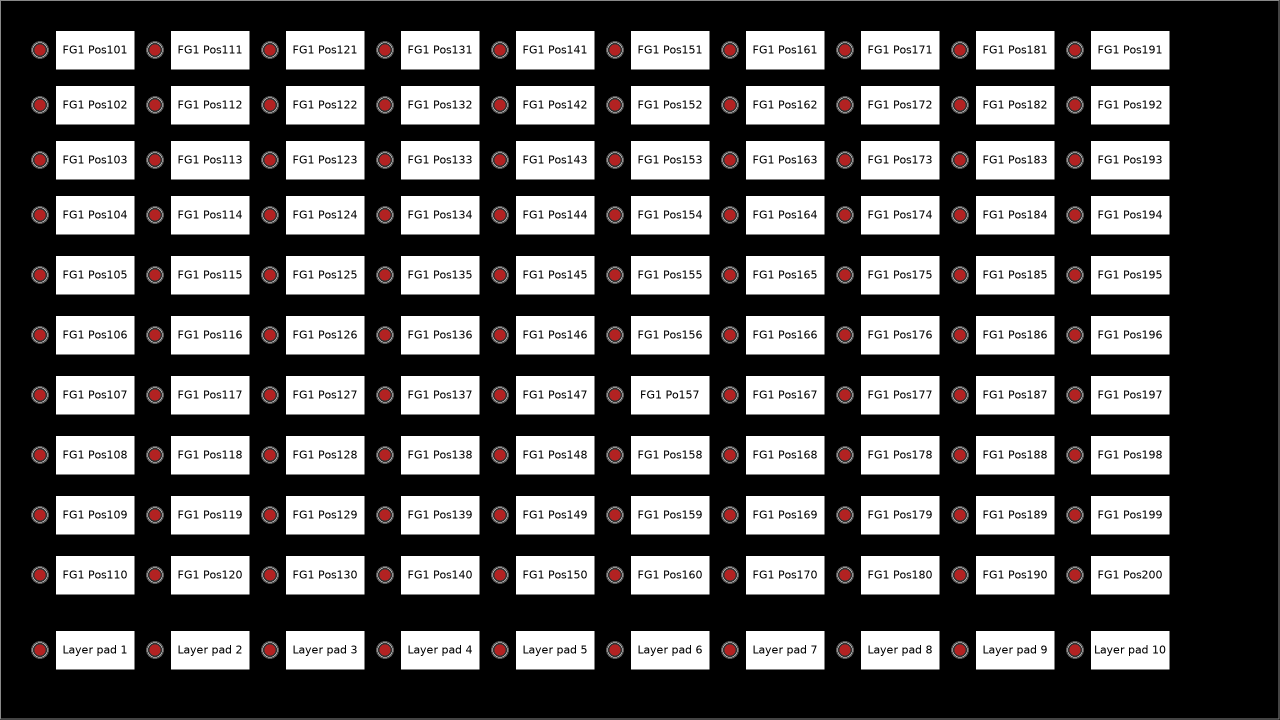
VISUALIZATION PAGE_KR1_Tab_1_200  // 1280x720
    RoundedRectangle (170,30 80x40), "FG1 Pos111"
        toggle KR1.bOutBit[18,0]
        OnMouseClick: execute {  }
    Lamp1 (145,40 20x20), variable: KR1.bInBit[18,0], style: Lamp-Lamp1-Red
    RoundedRectangle (55,30 80x40), "FG1 Pos101"
        toggle KR1.bOutBit[16,6]
        OnMouseClick: execute {  }
    Lamp1 (30,40 20x20), variable: KR1.bInBit[16,6], style: Lamp-Lamp1-Red
    RoundedRectangle (285,30 80x40), "FG1 Pos121"
        toggle KR1.bOutBit[19,2]
        OnMouseClick: execute {  }
    Lamp1 (260,40 20x20), variable: KR1.bInBit[19,2], style: Lamp-Lamp1-Red
    RoundedRectangle (400,30 80x40), "FG1 Pos131"
        toggle KR1.bOutBit[20,4]
        OnMouseClick: execute {  }
    Lamp1 (375,40 20x20), variable: KR1.bInBit[20,4], style: Lamp-Lamp1-Red
    RoundedRectangle (515,30 80x40), "FG1 Pos141"
        toggle KR1.bOutBit[21,6]
        OnMouseClick: execute {  }
    Lamp1 (490,40 20x20), variable: KR1.bInBit[21,6], style: Lamp-Lamp1-Red
    RoundedRectangle (745,30 80x40), "FG1 Pos161"
        toggle KR1.bOutBit[24,2]
        OnMouseClick: execute {  }
    Lamp1 (720,40 20x20), variable: KR1.bInBit[24,2], style: Lamp-Lamp1-Red
    RoundedRectangle (630,30 80x40), "FG1 Pos151"
        toggle KR1.bOutBit[23,0]
        OnMouseClick: execute {  }
    Lamp1 (605,40 20x20), variable: KR1.bInBit[23,0], style: Lamp-Lamp1-Red
    RoundedRectangle (860,30 80x40), "FG1 Pos171"
        toggle KR1.bOutBit[25,4]
        OnMouseClick: execute {  }
    Lamp1 (835,40 20x20), variable: KR1.bInBit[25,4], style: Lamp-Lamp1-Red
    RoundedRectangle (975,30 80x40), "FG1 Pos181"
        toggle KR1.bOutBit[26,6]
        OnMouseClick: execute {  }
    Lamp1 (950,40 20x20), variable: KR1.bInBit[26,6], style: Lamp-Lamp1-Red
    RoundedRectangle (1090,30 80x40), "FG1 Pos191"
        toggle KR1.bOutBit[28,0]
        OnMouseClick: execute {  }
    Lamp1 (1065,40 20x20), variable: KR1.bInBit[28,0], style: Lamp-Lamp1-Red
    RoundedRectangle (170,85 80x40), "FG1 Pos112"
        toggle KR1.bOutBit[18,1]
        OnMouseClick: execute {  }
    Lamp1 (145,95 20x20), variable: KR1.bInBit[18,1], style: Lamp-Lamp1-Red
    RoundedRectangle (55,85 80x40), "FG1 Pos102"
        toggle KR1.bOutBit[16,7]
        OnMouseClick: execute {  }
    Lamp1 (30,95 20x20), variable: KR1.bInBit[16,7], style: Lamp-Lamp1-Red
    RoundedRectangle (285,85 80x40), "FG1 Pos122"
        toggle KR1.bOutBit[19,3]
        OnMouseClick: execute {  }
    Lamp1 (260,95 20x20), variable: KR1.bInBit[19,3], style: Lamp-Lamp1-Red
    RoundedRectangle (400,85 80x40), "FG1 Pos132"
        toggle KR1.bOutBit[20,5]
        OnMouseClick: execute {  }
    Lamp1 (375,95 20x20), variable: KR1.bInBit[20,5], style: Lamp-Lamp1-Red
    RoundedRectangle (515,85 80x40), "FG1 Pos142"
        toggle KR1.bOutBit[21,7]
        OnMouseClick: execute {  }
    Lamp1 (490,95 20x20), variable: KR1.bInBit[21,7], style: Lamp-Lamp1-Red
    RoundedRectangle (745,85 80x40), "FG1 Pos162"
        toggle KR1.bOutBit[24,3]
        OnMouseClick: execute {  }
    Lamp1 (720,95 20x20), variable: KR1.bInBit[24,3], style: Lamp-Lamp1-Red
    RoundedRectangle (630,85 80x40), "FG1 Pos152"
        toggle KR1.bOutBit[23,1]
        OnMouseClick: execute {  }
    Lamp1 (605,95 20x20), variable: KR1.bInBit[23,1], style: Lamp-Lamp1-Red
    RoundedRectangle (860,85 80x40), "FG1 Pos172"
        toggle KR1.bOutBit[25,5]
        OnMouseClick: execute {  }
    Lamp1 (835,95 20x20), variable: KR1.bInBit[25,5], style: Lamp-Lamp1-Red
    RoundedRectangle (975,85 80x40), "FG1 Pos182"
        toggle KR1.bOutBit[26,7]
        OnMouseClick: execute {  }
    Lamp1 (950,95 20x20), variable: KR1.bInBit[26,7], style: Lamp-Lamp1-Red
    RoundedRectangle (1090,85 80x40), "FG1 Pos192"
        toggle KR1.bOutBit[28,1]
        OnMouseClick: execute {  }
    Lamp1 (1065,95 20x20), variable: KR1.bInBit[28,1], style: Lamp-Lamp1-Red
    RoundedRectangle (170,140 80x40), "FG1 Pos113"
        toggle KR1.bOutBit[18,2]
        OnMouseClick: execute {  }
    Lamp1 (145,150 20x20), variable: KR1.bInBit[18,2], style: Lamp-Lamp1-Red
    RoundedRectangle (55,140 80x40), "FG1 Pos103"
        toggle KR1.bOutBit[17,0]
        OnMouseClick: execute {  }
    Lamp1 (30,150 20x20), variable: KR1.bInBit[17,0], style: Lamp-Lamp1-Red
    RoundedRectangle (285,140 80x40), "FG1 Pos123"
        toggle KR1.bOutBit[19,4]
        OnMouseClick: execute {  }
    Lamp1 (260,150 20x20), variable: KR1.bInBit[19,4], style: Lamp-Lamp1-Red
    RoundedRectangle (400,140 80x40), "FG1 Pos133"
        toggle KR1.bOutBit[20,6]
        OnMouseClick: execute {  }
    Lamp1 (375,150 20x20), variable: KR1.bInBit[20,6], style: Lamp-Lamp1-Red
    RoundedRectangle (515,140 80x40), "FG1 Pos143"
        toggle KR1.bOutBit[22,0]
        OnMouseClick: execute {  }
    Lamp1 (490,150 20x20), variable: KR1.bInBit[22,0], style: Lamp-Lamp1-Red
    RoundedRectangle (745,140 80x40), "FG1 Pos163"
        toggle KR1.bOutBit[24,4]
        OnMouseClick: execute {  }
    Lamp1 (720,150 20x20), variable: KR1.bInBit[24,4], style: Lamp-Lamp1-Red
    RoundedRectangle (630,140 80x40), "FG1 Pos153"
        toggle KR1.bOutBit[23,2]
        OnMouseClick: execute {  }
    Lamp1 (605,150 20x20), variable: KR1.bInBit[23,2], style: Lamp-Lamp1-Red
    RoundedRectangle (860,140 80x40), "FG1 Pos173"
        toggle KR1.bOutBit[25,6]
        OnMouseClick: execute {  }
    Lamp1 (835,150 20x20), variable: KR1.bInBit[25,6], style: Lamp-Lamp1-Red
    RoundedRectangle (975,140 80x40), "FG1 Pos183"
        toggle KR1.bOutBit[27,0]
        OnMouseClick: execute {  }
    Lamp1 (950,150 20x20), variable: KR1.bInBit[27,0], style: Lamp-Lamp1-Red
    RoundedRectangle (1090,140 80x40), "FG1 Pos193"
        toggle KR1.bOutBit[28,2]
        OnMouseClick: execute {  }
    Lamp1 (1065,150 20x20), variable: KR1.bInBit[28,2], style: Lamp-Lamp1-Red
    RoundedRectangle (170,195 80x40), "FG1 Pos114"
        toggle KR1.bOutBit[18,3]
        OnMouseClick: execute {  }
    Lamp1 (145,205 20x20), variable: KR1.bInBit[18,3], style: Lamp-Lamp1-Red
    RoundedRectangle (55,195 80x40), "FG1 Pos104"
        toggle KR1.bOutBit[17,1]
        OnMouseClick: execute {  }
    Lamp1 (30,205 20x20), variable: KR1.bInBit[17,1], style: Lamp-Lamp1-Red
    RoundedRectangle (285,195 80x40), "FG1 Pos124"
        toggle KR1.bOutBit[19,5]
        OnMouseClick: execute {  }
    Lamp1 (260,205 20x20), variable: KR1.bInBit[19,5], style: Lamp-Lamp1-Red
    RoundedRectangle (400,195 80x40), "FG1 Pos134"
        toggle KR1.bOutBit[20,7]
        OnMouseClick: execute {  }
    Lamp1 (375,205 20x20), variable: KR1.bInBit[20,7], style: Lamp-Lamp1-Red
    RoundedRectangle (515,195 80x40), "FG1 Pos144"
        toggle KR1.bOutBit[22,1]
        OnMouseClick: execute {  }
    Lamp1 (490,205 20x20), variable: KR1.bInBit[22,1], style: Lamp-Lamp1-Red
    RoundedRectangle (745,195 80x40), "FG1 Pos164"
        toggle KR1.bOutBit[24,5]
        OnMouseClick: execute {  }
    Lamp1 (720,205 20x20), variable: KR1.bInBit[24,5], style: Lamp-Lamp1-Red
    RoundedRectangle (630,195 80x40), "FG1 Pos154"
        toggle KR1.bOutBit[23,3]
        OnMouseClick: execute {  }
    Lamp1 (605,205 20x20), variable: KR1.bInBit[23,3], style: Lamp-Lamp1-Red
    RoundedRectangle (860,195 80x40), "FG1 Pos174"
        toggle KR1.bOutBit[25,7]
        OnMouseClick: execute {  }
    Lamp1 (835,205 20x20), variable: KR1.bInBit[25,7], style: Lamp-Lamp1-Red
    RoundedRectangle (975,195 80x40), "FG1 Pos184"
        toggle KR1.bOutBit[27,1]
        OnMouseClick: execute {  }
    Lamp1 (950,205 20x20), variable: KR1.bInBit[27,1], style: Lamp-Lamp1-Red
    RoundedRectangle (1090,195 80x40), "FG1 Pos194"
        toggle KR1.bOutBit[28,3]
        OnMouseClick: execute {  }
    Lamp1 (1065,205 20x20), variable: KR1.bInBit[28,3], style: Lamp-Lamp1-Red
    RoundedRectangle (170,255 80x40), "FG1 Pos115"
        toggle KR1.bOutBit[18,4]
        OnMouseClick: execute {  }
    Lamp1 (145,265 20x20), variable: KR1.bInBit[18,4], style: Lamp-Lamp1-Red
    RoundedRectangle (55,255 80x40), "FG1 Pos105"
        toggle KR1.bOutBit[17,2]
        OnMouseClick: execute {  }
    Lamp1 (30,265 20x20), variable: KR1.bInBit[17,2], style: Lamp-Lamp1-Red
    RoundedRectangle (285,255 80x40), "FG1 Pos125"
        toggle KR1.bOutBit[19,6]
        OnMouseClick: execute {  }
    Lamp1 (260,265 20x20), variable: KR1.bInBit[19,6], style: Lamp-Lamp1-Red
    RoundedRectangle (400,255 80x40), "FG1 Pos135"
        toggle KR1.bOutBit[21,0]
        OnMouseClick: execute {  }
    Lamp1 (375,265 20x20), variable: KR1.bInBit[21,0], style: Lamp-Lamp1-Red
    RoundedRectangle (515,255 80x40), "FG1 Pos145"
        toggle KR1.bOutBit[22,2]
        OnMouseClick: execute {  }
    Lamp1 (490,265 20x20), variable: KR1.bInBit[22,2], style: Lamp-Lamp1-Red
    RoundedRectangle (745,255 80x40), "FG1 Pos165"
        toggle KR1.bOutBit[24,6]
        OnMouseClick: execute {  }
    Lamp1 (720,265 20x20), variable: KR1.bInBit[24,6], style: Lamp-Lamp1-Red
    RoundedRectangle (630,255 80x40), "FG1 Pos155"
        toggle KR1.bOutBit[23,4]
        OnMouseClick: execute {  }
    Lamp1 (605,265 20x20), variable: KR1.bInBit[23,4], style: Lamp-Lamp1-Red
    RoundedRectangle (860,255 80x40), "FG1 Pos175"
        toggle KR1.bOutBit[26,0]
        OnMouseClick: execute {  }
    Lamp1 (835,265 20x20), variable: KR1.bInBit[26,0], style: Lamp-Lamp1-Red
    RoundedRectangle (975,255 80x40), "FG1 Pos185"
        toggle KR1.bOutBit[27,2]
        OnMouseClick: execute {  }
    Lamp1 (950,265 20x20), variable: KR1.bInBit[27,2], style: Lamp-Lamp1-Red
    RoundedRectangle (1090,255 80x40), "FG1 Pos195"
        toggle KR1.bOutBit[28,4]
        OnMouseClick: execute {  }
    Lamp1 (1065,265 20x20), variable: KR1.bInBit[28,4], style: Lamp-Lamp1-Red
    RoundedRectangle (170,315 80x40), "FG1 Pos116"
        toggle KR1.bOutBit[18,5]
        OnMouseClick: execute {  }
    Lamp1 (145,325 20x20), variable: KR1.bInBit[18,5], style: Lamp-Lamp1-Red
    RoundedRectangle (55,315 80x40), "FG1 Pos106"
        toggle KR1.bOutBit[17,3]
        OnMouseClick: execute {  }
    Lamp1 (30,325 20x20), variable: KR1.bInBit[17,3], style: Lamp-Lamp1-Red
    RoundedRectangle (285,315 80x40), "FG1 Pos126"
        toggle KR1.bOutBit[19,7]
        OnMouseClick: execute {  }
    Lamp1 (260,325 20x20), variable: KR1.bInBit[19,7], style: Lamp-Lamp1-Red
    RoundedRectangle (400,315 80x40), "FG1 Pos136"
        toggle KR1.bOutBit[21,1]
        OnMouseClick: execute {  }
    Lamp1 (375,325 20x20), variable: KR1.bInBit[21,1], style: Lamp-Lamp1-Red
    RoundedRectangle (515,315 80x40), "FG1 Pos146"
        toggle KR1.bOutBit[22,3]
        OnMouseClick: execute {  }
    Lamp1 (490,325 20x20), variable: KR1.bInBit[22,3], style: Lamp-Lamp1-Red
    RoundedRectangle (745,315 80x40), "FG1 Pos166"
        toggle KR1.bOutBit[24,7]
        OnMouseClick: execute {  }
    Lamp1 (720,325 20x20), variable: KR1.bInBit[24,7], style: Lamp-Lamp1-Red
    RoundedRectangle (630,315 80x40), "FG1 Pos156"
        toggle KR1.bOutBit[23,5]
        OnMouseClick: execute {  }
    Lamp1 (605,325 20x20), variable: KR1.bInBit[23,5], style: Lamp-Lamp1-Red
    RoundedRectangle (860,315 80x40), "FG1 Pos176"
        toggle KR1.bOutBit[26,1]
        OnMouseClick: execute {  }
    Lamp1 (835,325 20x20), variable: KR1.bInBit[26,1], style: Lamp-Lamp1-Red
    RoundedRectangle (975,315 80x40), "FG1 Pos186"
        toggle KR1.bOutBit[27,3]
        OnMouseClick: execute {  }
    Lamp1 (950,325 20x20), variable: KR1.bInBit[27,3], style: Lamp-Lamp1-Red
    RoundedRectangle (1090,315 80x40), "FG1 Pos196"
        toggle KR1.bOutBit[28,5]
        OnMouseClick: execute {  }
    Lamp1 (1065,325 20x20), variable: KR1.bInBit[28,5], style: Lamp-Lamp1-Red
    RoundedRectangle (170,375 80x40), "FG1 Pos117"
        toggle KR1.bOutBit[18,6]
        OnMouseClick: execute {  }
    Lamp1 (145,385 20x20), variable: KR1.bInBit[18,6], style: Lamp-Lamp1-Red
    RoundedRectangle (55,375 80x40), "FG1 Pos107"
        toggle KR1.bOutBit[17,4]
        OnMouseClick: execute {  }
    Lamp1 (30,385 20x20), variable: KR1.bInBit[17,4], style: Lamp-Lamp1-Red
    RoundedRectangle (285,375 80x40), "FG1 Pos127"
        toggle KR1.bOutBit[20,0]
        OnMouseClick: execute {  }
    Lamp1 (260,385 20x20), variable: KR1.bInBit[20,0], style: Lamp-Lamp1-Red
    RoundedRectangle (400,375 80x40), "FG1 Pos137"
        toggle KR1.bOutBit[21,2]
        OnMouseClick: execute {  }
    Lamp1 (375,385 20x20), variable: KR1.bInBit[21,2], style: Lamp-Lamp1-Red
    RoundedRectangle (515,375 80x40), "FG1 Pos147"
        toggle KR1.bOutBit[22,4]
        OnMouseClick: execute {  }
    Lamp1 (490,385 20x20), variable: KR1.bInBit[22,4], style: Lamp-Lamp1-Red
    RoundedRectangle (745,375 80x40), "FG1 Pos167"
        toggle KR1.bOutBit[25,0]
        OnMouseClick: execute {  }
    Lamp1 (720,385 20x20), variable: KR1.bInBit[25,0], style: Lamp-Lamp1-Red
    RoundedRectangle (630,375 80x40), "FG1 Po157"
        toggle KR1.bOutBit[23,6]
        OnMouseClick: execute {  }
    Lamp1 (605,385 20x20), variable: KR1.bInBit[23,6], style: Lamp-Lamp1-Red
    RoundedRectangle (860,375 80x40), "FG1 Pos177"
        toggle KR1.bOutBit[26,2]
        OnMouseClick: execute {  }
    Lamp1 (835,385 20x20), variable: KR1.bInBit[26,2], style: Lamp-Lamp1-Red
    RoundedRectangle (975,375 80x40), "FG1 Pos187"
        toggle KR1.bOutBit[27,4]
        OnMouseClick: execute {  }
    Lamp1 (950,385 20x20), variable: KR1.bInBit[27,4], style: Lamp-Lamp1-Red
    RoundedRectangle (1090,375 80x40), "FG1 Pos197"
        toggle KR1.bOutBit[28,6]
        OnMouseClick: execute {  }
    Lamp1 (1065,385 20x20), variable: KR1.bInBit[28,6], style: Lamp-Lamp1-Red
    RoundedRectangle (170,435 80x40), "FG1 Pos118"
        toggle KR1.bOutBit[18,7]
        OnMouseClick: execute {  }
    Lamp1 (145,445 20x20), variable: KR1.bInBit[18,7], style: Lamp-Lamp1-Red
    RoundedRectangle (55,435 80x40), "FG1 Pos108"
        toggle KR1.bOutBit[17,5]
        OnMouseClick: execute {  }
    Lamp1 (30,445 20x20), variable: KR1.bInBit[17,5], style: Lamp-Lamp1-Red
    RoundedRectangle (285,435 80x40), "FG1 Pos128"
        toggle KR1.bOutBit[20,1]
        OnMouseClick: execute {  }
    Lamp1 (260,445 20x20), variable: KR1.bInBit[20,1], style: Lamp-Lamp1-Red
    RoundedRectangle (400,435 80x40), "FG1 Pos138"
        toggle KR1.bOutBit[21,3]
        OnMouseClick: execute {  }
    Lamp1 (375,445 20x20), variable: KR1.bInBit[21,3], style: Lamp-Lamp1-Red
    RoundedRectangle (515,435 80x40), "FG1 Pos148"
        toggle KR1.bOutBit[22,5]
        OnMouseClick: execute {  }
    Lamp1 (490,445 20x20), variable: KR1.bInBit[22,5], style: Lamp-Lamp1-Red
    RoundedRectangle (745,435 80x40), "FG1 Pos168"
        toggle KR1.bOutBit[25,1]
        OnMouseClick: execute {  }
    Lamp1 (720,445 20x20), variable: KR1.bInBit[25,1], style: Lamp-Lamp1-Red
    RoundedRectangle (630,435 80x40), "FG1 Pos158"
        toggle KR1.bOutBit[23,7]
        OnMouseClick: execute {  }
    Lamp1 (605,445 20x20), variable: KR1.bInBit[23,7], style: Lamp-Lamp1-Red
    RoundedRectangle (860,435 80x40), "FG1 Pos178"
        toggle KR1.bOutBit[26,3]
        OnMouseClick: execute {  }
    Lamp1 (835,445 20x20), variable: KR1.bInBit[26,3], style: Lamp-Lamp1-Red
    RoundedRectangle (975,435 80x40), "FG1 Pos188"
        toggle KR1.bOutBit[27,5]
        OnMouseClick: execute {  }
    Lamp1 (950,445 20x20), variable: KR1.bInBit[27,5], style: Lamp-Lamp1-Red
    RoundedRectangle (1090,435 80x40), "FG1 Pos198"
        toggle KR1.bOutBit[28,7]
        OnMouseClick: execute {  }
    Lamp1 (1065,445 20x20), variable: KR1.bInBit[28,7], style: Lamp-Lamp1-Red
    RoundedRectangle (55,495 80x40), "FG1 Pos109"
        toggle KR1.bOutBit[17,6]
        OnMouseClick: execute {  }
    Lamp1 (30,505 20x20), variable: KR1.bInBit[17,6], style: Lamp-Lamp1-Red
    RoundedRectangle (170,495 80x40), "FG1 Pos119"
        toggle KR1.bOutBit[19,0]
        OnMouseClick: execute {  }
    Lamp1 (145,505 20x20), variable: KR1.bInBit[19,0], style: Lamp-Lamp1-Red
    RoundedRectangle (285,495 80x40), "FG1 Pos129"
        toggle KR1.bOutBit[20,2]
        OnMouseClick: execute {  }
    Lamp1 (260,505 20x20), variable: KR1.bInBit[20,2], style: Lamp-Lamp1-Red
    RoundedRectangle (400,495 80x40), "FG1 Pos139"
        toggle KR1.bOutBit[21,4]
        OnMouseClick: execute {  }
    Lamp1 (375,505 20x20), variable: KR1.bInBit[21,4], style: Lamp-Lamp1-Red
    RoundedRectangle (515,495 80x40), "FG1 Pos149"
        toggle KR1.bOutBit[22,6]
        OnMouseClick: execute {  }
    Lamp1 (490,505 20x20), variable: KR1.bInBit[22,6], style: Lamp-Lamp1-Red
    RoundedRectangle (630,495 80x40), "FG1 Pos159"
        toggle KR1.bOutBit[24,0]
        OnMouseClick: execute {  }
    Lamp1 (605,505 20x20), variable: KR1.bInBit[24,0], style: Lamp-Lamp1-Red
    RoundedRectangle (745,495 80x40), "FG1 Pos169"
        toggle KR1.bOutBit[25,2]
        OnMouseClick: execute {  }
    Lamp1 (720,505 20x20), variable: KR1.bInBit[25,2], style: Lamp-Lamp1-Red
    RoundedRectangle (860,495 80x40), "FG1 Pos179"
        toggle KR1.bOutBit[26,4]
        OnMouseClick: execute {  }
    Lamp1 (835,505 20x20), variable: KR1.bInBit[26,4], style: Lamp-Lamp1-Red
    RoundedRectangle (975,495 80x40), "FG1 Pos189"
        toggle KR1.bOutBit[27,6]
        OnMouseClick: execute {  }
    Lamp1 (950,505 20x20), variable: KR1.bInBit[27,6], style: Lamp-Lamp1-Red
    RoundedRectangle (1090,495 80x40), "FG1 Pos199"
        toggle KR1.bOutBit[29,0]
        OnMouseClick: execute {  }
    Lamp1 (1065,505 20x20), variable: KR1.bInBit[29,0], style: Lamp-Lamp1-Red
    RoundedRectangle (55,555 80x40), "FG1 Pos110"
        toggle KR1.bOutBit[17,7]
        OnMouseClick: execute {  }
    Lamp1 (30,565 20x20), variable: KR1.bInBit[17,7], style: Lamp-Lamp1-Red
    RoundedRectangle (170,555 80x40), "FG1 Pos120"
        toggle KR1.bOutBit[19,1]
        OnMouseClick: execute {  }
    Lamp1 (145,565 20x20), variable: KR1.bInBit[19,1], style: Lamp-Lamp1-Red
    RoundedRectangle (285,555 80x40), "FG1 Pos130"
        toggle KR1.bOutBit[20,3]
        OnMouseClick: execute {  }
    Lamp1 (260,565 20x20), variable: KR1.bInBit[20,3], style: Lamp-Lamp1-Red
    RoundedRectangle (400,555 80x40), "FG1 Pos140"
        toggle KR1.bOutBit[21,5]
        OnMouseClick: execute {  }
    Lamp1 (375,565 20x20), variable: KR1.bInBit[21,5], style: Lamp-Lamp1-Red
    RoundedRectangle (515,555 80x40), "FG1 Pos150"
        toggle KR1.bOutBit[22,7]
        OnMouseClick: execute {  }
    Lamp1 (490,565 20x20), variable: KR1.bInBit[22,7], style: Lamp-Lamp1-Red
    RoundedRectangle (630,555 80x40), "FG1 Pos160"
        toggle KR1.bOutBit[24,1]
        OnMouseClick: execute {  }
    Lamp1 (605,565 20x20), variable: KR1.bInBit[24,1], style: Lamp-Lamp1-Red
    RoundedRectangle (745,555 80x40), "FG1 Pos170"
        toggle KR1.bOutBit[25,3]
        OnMouseClick: execute {  }
    Lamp1 (720,565 20x20), variable: KR1.bInBit[25,3], style: Lamp-Lamp1-Red
    RoundedRectangle (860,555 80x40), "FG1 Pos180"
        toggle KR1.bOutBit[26,5]
        OnMouseClick: execute {  }
    Lamp1 (835,565 20x20), variable: KR1.bInBit[26,5], style: Lamp-Lamp1-Red
    RoundedRectangle (975,555 80x40), "FG1 Pos190"
        toggle KR1.bOutBit[27,7]
        OnMouseClick: execute {  }
    Lamp1 (950,565 20x20), variable: KR1.bInBit[27,7], style: Lamp-Lamp1-Red
    RoundedRectangle (1090,555 80x40), "FG1 Pos200"
        toggle KR1.bOutBit[29,1]
        OnMouseClick: execute {  }
    Lamp1 (1065,565 20x20), variable: KR1.bInBit[29,1], style: Lamp-Lamp1-Red
    RoundedRectangle (55,630 80x40), "Layer pad 1"
        toggle KR1.bOutBit[29,2]
        OnMouseClick: execute {  }
    Lamp1 (30,640 20x20), variable: KR1.bInBit[29,2], style: Lamp-Lamp1-Red
    RoundedRectangle (170,630 80x40), "Layer pad 2"
        toggle KR1.bOutBit[29,3]
        OnMouseClick: execute {  }
    Lamp1 (145,640 20x20), variable: KR1.bInBit[29,3], style: Lamp-Lamp1-Red
    RoundedRectangle (285,630 80x40), "Layer pad 3"
        toggle KR1.bOutBit[29,4]
        OnMouseClick: execute {  }
    Lamp1 (260,640 20x20), variable: KR1.bInBit[29,4], style: Lamp-Lamp1-Red
    RoundedRectangle (400,630 80x40), "Layer pad 4"
        toggle KR1.bOutBit[29,5]
        OnMouseClick: execute {  }
    Lamp1 (375,640 20x20), variable: KR1.bInBit[29,5], style: Lamp-Lamp1-Red
    RoundedRectangle (515,630 80x40), "Layer pad 5"
        toggle KR1.bOutBit[29,6]
        OnMouseClick: execute {  }
    Lamp1 (490,640 20x20), variable: KR1.bInBit[29,6], style: Lamp-Lamp1-Red
    RoundedRectangle (630,630 80x40), "Layer pad 6"
        toggle KR1.bOutBit[29,7]
        OnMouseClick: execute {  }
    Lamp1 (605,640 20x20), variable: KR1.bInBit[29,7], style: Lamp-Lamp1-Red
    RoundedRectangle (745,630 80x40), "Layer pad 7"
        toggle KR1.bOutBit[30,0]
        OnMouseClick: execute {  }
    Lamp1 (720,640 20x20), variable: KR1.bInBit[30,0], style: Lamp-Lamp1-Red
    RoundedRectangle (860,630 80x40), "Layer pad 8"
        toggle KR1.bOutBit[30,1]
        OnMouseClick: execute {  }
    Lamp1 (835,640 20x20), variable: KR1.bInBit[30,1], style: Lamp-Lamp1-Red
    RoundedRectangle (975,630 80x40), "Layer pad 9"
        toggle KR1.bOutBit[30,2]
        OnMouseClick: execute {  }
    Lamp1 (950,640 20x20), variable: KR1.bInBit[30,2], style: Lamp-Lamp1-Red
    RoundedRectangle (1090,630 80x40), "Layer pad 10"
        toggle KR1.bOutBit[30,3]
        OnMouseClick: execute {  }
    Lamp1 (1065,640 20x20), variable: KR1.bInBit[30,3], style: Lamp-Lamp1-Red
END_VISUALIZATION

(* stored: Version 1.1.0.1, ProductVersion 3.1.4024.12
   Visu PAGE_KR1_Tab_1_200: Id {b49f1993-61de-4574-8724-c338c6975e7c} *)
